// TIA Portal V18 export
// export: Created 2025-12-01T12:38:49.5591989Z, ExportSetting None, DisplayName Totally Integrated Automation Portal, DisplayVersion V18 Update 5, DisplayName TIA Portal Openness, DisplayVersion V18 Update 5, DisplayName TIA Portal Teamcenter Gateway, DisplayVersion V18, DisplayName TIA Portal Version Control Interface, DisplayVersion V18, DisplayName STEP 7 Professional, DisplayVersion V18 Update 5, DisplayName STEP 7 Safety, DisplayVersion V18, DisplayName WinCC Professional, DisplayVersion V18 Update 5
DATA_BLOCK "GluingControl"   // DB2800
{ S7_Optimized_Access := 'FALSE' }
// stored: AutoNumber false
   VAR
      Input : Struct
         GluingDeviceReady : Bool;
         GluingFault : Bool;
         GluingRefillTank : Bool;
         GluingTankEmpty : Bool;
      END_STRUCT;
      Output : Struct
         GluingPro_X : Bool;
         GluingPro_Y : Bool;
         GluingPro_Z : Bool;
         GluingReset : Bool;
      END_STRUCT;
      Control : Struct
         Manual_X : Bool;
         Manual_Y : Bool;
         Manual_Z : Bool;
         Manual_Control : Int;
         Auto_Start : Bool;
         Auto_Y : Bool;
         Auto_Z : Bool;
         Auto_Control : Int;
         ManualTest_X : Bool;
         ManualTestStartGlue : Bool;
      END_STRUCT;
      GlueCalibratonMode : Bool;
      TON : Array[1..10] of IEC_LTIMER;
      P { S7_SetPoint := 'True'} : Array[1..10] of Bool;
      GlueInitiaStart : Bool;
   END_VAR
BEGIN
END_DATA_BLOCK
